// TwinCAT 3 PLC project PLC
// ProgramVersion: 3.1.4024.0
// libraries:
//   Tc2_Standard, * (Beckhoff Automation GmbH)
//   Tc2_System, * (Beckhoff Automation GmbH)
//   Tc3_Module, * (Beckhoff Automation GmbH)
// project tree:
//   DUTs/ FixtureInput.TcDUT, FixtureOutput.TcDUT, RollerDoor.TcDUT, Turn.TcDUT, TurnTableOutput.TcDUT
//   DUTs/Robot/ udt_HDL_CellToHandling.TcDUT, udt_HDL_HandlingToCell.TcDUT, udt_HDL_PartData.TcDUT
//   / GlobalTextList.TcGTLO, PlcTask.TcTTO, Visualization Manager.TcVMO (not stored)
//   GVLs/ IO.TcGVL, Memory.TcGVL, HMI.TcGVL, RobotInterface.TcGVL, WeldRobotInterface.TcGVL
//   POUs/ AutoSequence.TcPOU, Call_Fb.TcPOU, Feedback.TcPOU, Clamping.TcPOU, MAIN.TcPOU, RobotMH.TcPOU, RoolerDoor.TcPOU, Turn_Table.TcPOU, Turning_fb.TcPOU, vishalTest.TcPOU, WeldRobot.TcPOU
//   VISUs/ Clamp.TcVIS
// real-time tasks:
//   TASK PlcTask: cycle T#10ms, priority 20, ADS port 350

CONFIGURATION PLC
    RESOURCE PLC ON TwinCAT3
        TASK PlcTask(INTERVAL := T#10ms, PRIORITY := 20);
        PROGRAM MAIN WITH PlcTask : MAIN;
    END_RESOURCE
END_CONFIGURATION

// ---- DUTs/FixtureInput.TcDUT
TYPE FixtureInput :
STRUCT
i_Control_Pressure_Sw_In1_BPB1:BOOL;
i_Control_Pressure_Sw_In2_BPB1:BOOL;
i_Valve_Pos_BGB1:BOOL;
i_Reserve_BPB1_0_3:BOOL;
i_CC6_Clamp_1_Sensor_HP:BOOL;
i_CC6_Clamp_1_Sensor_WP:BOOL;
i_CC4_Clamp_3_Sensor_HP:BOOL;
i_CC4_Clamp_3_Sensor_WP:BOOL;
i_PART_CONTROL_B13:BOOL;
i_PART_CONTROL_B27:BOOL;
i_PART_CONTROL_B14:BOOL;
i_PART_CONTROL_B28:BOOL;
i_Reserve_BGB1_1_4:BOOL;
i_Reserve_BGB1_1_5:BOOL;

i_Reserve_2_0:BOOL;
i_Reserve_2_1:BOOL;
i_Reserve_2_2:BOOL;
i_Reserve_2_3:BOOL;
i_Reserve_2_4:BOOL;
i_Reserve_2_5:BOOL;
i_Reserve_2_6:BOOL;
i_Reserve_2_7:BOOL;
i_Reserve_3_0:BOOL;
i_Reserve_3_1:BOOL;
i_Reserve_3_2:BOOL;
i_Reserve_3_3:BOOL;
i_Reserve_3_4:BOOL;
i_Reserve_3_5:BOOL;
i_Reserve_3_6:BOOL;
i_Reserve_3_7:BOOL;
i_CC4_Clamp_2_Sensor_HP:BOOL;
i_CC4_Clamp_2_Sensor_WP:BOOL;
i_CC4_Clamp_1_Sensor_HP:BOOL;
i_CC4_Clamp_1_Sensor_WP:BOOL;
i_CC2_Clamp_3_Sensor_HP:BOOL;
i_CC2_Clamp_3_Sensor_WP:BOOL;
i_PART_CONTROL_B12:BOOL;
i_PART_CONTROL_B26:BOOL;
i_PART_CONTROL_B11:BOOL;
i_PART_CONTROL_B25:BOOL;
i_PART_CONTROL_B10:BOOL;
i_PART_CONTROL_B24:BOOL;
i_Reserve_5_4:BOOL;
i_Reserve_5_5:BOOL;
i_Reserve_5_6:BOOL;
i_Reserve_5_7:BOOL;
i_Reserve_6_0:BOOL;
i_Reserve_6_1:BOOL;
i_Reserve_6_2:BOOL;
i_Reserve_6_3:BOOL;
i_Reserve_6_4:BOOL;
i_Reserve_6_5:BOOL;
i_Reserve_6_6:BOOL;
i_Reserve_6_7:BOOL;
i_Reserve_7_1:BOOL;
i_Reserve_7_2:BOOL;
i_Reserve_7_3:BOOL;
i_Reserve_7_4:BOOL;
i_Reserve_7_5:BOOL;
i_Reserve_7_6:BOOL;
i_Reserve_7_7:BOOL;
i_CC3_Clamp_3_Sensor_HP:BOOL;
i_CC3_Clamp_3_Sensor_WP:BOOL;
i_CC3_Clamp_2_Sensor_HP:BOOL;
i_CC3_Clamp_2_Sensor_WP:BOOL;
i_CC3_Clamp_1_Sensor_HP:BOOL;
i_CC3_Clamp_1_Sensor_WP:BOOL;
i_PART_CONTROL_B7:BOOL;
i_PART_CONTROL_B21:BOOL;
i_PART_CONTROL_B6:BOOL;
i_PART_CONTROL_B20:BOOL;
i_PART_CONTROL_B5:BOOL;
i_PART_CONTROL_B19:BOOL;
i_Reserve_9_4:BOOL;
i_Reserve_9_5:BOOL;

i_CC1_Clamp_3_Sensor_HP:BOOL;
i_CC1_Clamp_3_Sensor_WP:BOOL;
i_CC1_Clamp_2_Sensor_HP:BOOL;
i_CC1_Clamp_2_Sensor_WP:BOOL;
i_CC1_Clamp_1_Sensor_HP:BOOL;
i_CC1_Clamp_1_Sensor_WP:BOOL;
i_PART_CONTROL_B4:BOOL;
i_PART_CONTROL_B18:BOOL;
i_PART_CONTROL_B3:BOOL;
i_PART_CONTROL_B17:BOOL;
i_PART_CONTROL_B2:BOOL;
i_PART_CONTROL_B16:BOOL;

i_CC2_Clamp_2_Sensor_HP:BOOL;
i_CC2_Clamp_2_Sensor_WP:BOOL;
i_CC2_Clamp_1_Sensor_HP:BOOL;
i_CC2_Clamp_1_Sensor_WP:BOOL;
i_PART_CONTROL_B9:BOOL;
i_PART_CONTROL_B23:BOOL;
i_PART_CONTROL_B8:BOOL;
i_PART_CONTROL_B22:BOOL;

i_CC5_Clamp_1_Sensor_HP:BOOL;
i_CC5_Clamp_1_Sensor_WP:BOOL;
i_PART_CONTROL_B1:BOOL;
i_PART_CONTROL_B15:BOOL;



END_STRUCT
END_TYPE

// ---- DUTs/FixtureOutput.TcDUT
TYPE FixtureOutput :
STRUCT
	o_CC1_CLAMPING_UNIT1_3_WP:BOOL;
o_CC1_CLAMPING_UNIT1_3_HP:BOOL;
o_CC2_CLAMPING_UNIT2_3_WP:BOOL;
o_CC2_CLAMPING_UNIT2_3_HP:BOOL;
o_CC3_CLAMPING_UNIT3_3_WP:BOOL;
o_CC3_CLAMPING_UNIT3_3_HP:BOOL;
o_CC4_CLAMPING_UNIT4_3_WP:BOOL;
o_CC4_CLAMPING_UNIT4_3_HP:BOOL;
o_CC5_CLAMPING_UNIT5_1_WP:BOOL;
o_CC5_CLAMPING_UNIT5_1_HP:BOOL;
o_CC6_CLAMPING_UNIT6_1_WP:BOOL;
o_CC6_CLAMPING_UNIT6_1_HP:BOOL;
o_RESERVE_1_4:BOOL;
o_RESERVE_1_5:BOOL;
o_RESERVE_1_6:BOOL;
o_RESERVE_1_7:BOOL;
o_RESERVE_2_0:BOOL;
o_RESERVE_2_1:BOOL;
o_RESERVE_2_2:BOOL;
o_RESERVE_2_3:BOOL;
o_RESERVE_2_4:BOOL;
o_RESERVE_2_5:BOOL;
o_RESERVE_2_6:BOOL;
o_RESERVE_2_7:BOOL;
o_RESERVE_3_0:BOOL;
o_RESERVE_3_1:BOOL;
o_RESERVE_3_2:BOOL;
o_RESERVE_3_3:BOOL;
o_RESERVE_3_4:BOOL;
o_RESERVE_3_5:BOOL;
o_RESERVE_3_6:BOOL;
o_RESERVE_3_7:BOOL;

END_STRUCT
END_TYPE

// ---- DUTs/Robot/udt_HDL_CellToHandling.TcDUT
TYPE udt_HDL_CellToHandling :
STRUCT
    (* Cell state *)
    Status      : WORD; // 0: Auto, 2: Manual, 3: Error
    Time_Stamp  : DATE_AND_TIME;
    part        : udt_HDL_PartData; // part
    
    (* Job Handshake *)
    Request             : USINT; // 20: Pick, 10: Drop
    RequestPartType     : BOOL;
    GateOpened          : BOOL;
    GateClosed          : BOOL;
    FixtureReady        : BOOL;
    (* Progress Feedback *)
	RaiseEnable1        : BOOL;
    RaiseEnable2        : BOOL;
    ReduceEnable1       : BOOL;
    ReduceEnable2       : BOOL;
     (* Status/Confirmation *)
	PickJobAck          : BOOL;
    DropJobAck          : BOOL;
    Hold                : BOOL;
    (* Gripper Acknowledge *)
	Gripper1ReadyToClose : BOOL;
    Gripper1ReadyToOpen  : BOOL;
    Gripper2ReadyToClose : BOOL;
    Gripper2ReadyToOpen  : BOOL;
    FeatureBit6         : BOOL;
    FeatureBit7         : BOOL;
END_STRUCT
END_TYPE

// ---- DUTs/Robot/udt_HDL_HandlingToCell.TcDUT
TYPE udt_HDL_HandlingToCell :
STRUCT
	
(* HDL Data *)
    Status      : WORD; // 0 Auto -- 1 Auto Startup -- 2 Manual -- 3 Error -- 4 LineMode -- 5 PowerOn -- 6 EnergySave -- 7 SafeOk
    part        : udt_HDL_PartData; // part
    
    (* Job Handshake Requests & Logic *)
    GateOpenRequest     : BOOL;
    GateCloseRequest    : BOOL;
    PickJobProceed      : BOOL;
    DropJobProceed      : BOOL;
    
    (* Progress Feedback *)
    RaiseFinished1      : BOOL;
    RaiseFinished2      : BOOL;
    ReduceFinished1     : BOOL;
    ReduceFinished2     : BOOL;
    
    (* Status/Confirmation *)
    PickJobOK           : BOOL;
    DropJobOK           : BOOL;
    InArea              : BOOL;
    PickDropProceed     : BOOL;
    
    (* Gripper Acknowledge *)
    Gripper1ClosedAck   : BOOL;
    Gripper1OpenedAck   : BOOL;
    Gripper2ClosedAck   : BOOL;
    Gripper2OpenedAck   : BOOL;
    
    (* Spare/Auxiliary *)
    FeatureBit6         : BOOL;
    FeatureBit7         : BOOL;
    PickEnable          : BOOL;
    DropEnable          : BOOL;
    
    (* Process Data *)
    Types               : USINT;
    ActiveCell          : USINT;
    Cooling_Time_Buffer : DINT;
    FB_Cooling_Time     : DINT;
END_STRUCT
END_TYPE

// ---- DUTs/Robot/udt_HDL_PartData.TcDUT
TYPE udt_HDL_PartData :
STRUCT
PartId	:DINT; //Unique Part Id (DMC Serial Number)
State	:BOOL; //Part state 0=OK, 1=NOK
Types :	BOOL;// Part type 1=Long, 0=Short
Exists	:BOOL; //Part exist


END_STRUCT
END_TYPE

// ---- DUTs/RollerDoor.TcDUT
TYPE RollerDoor :
STRUCT
	
i_RD_Sensor_Open:BOOL;
i_RD_Sensor_Close:BOOL;
o_RD_Open:BOOL;
o_RD_Close:BOOL;

END_STRUCT
END_TYPE

// ---- DUTs/Turn.TcDUT
TYPE Turn :
STRUCT
	o_Turn_REF_SENSOR:BOOL;
o_Turn_FWD_SENSOR:BOOL;
o_Turn_REV_SENSOR:BOOL;
END_STRUCT
END_TYPE

// ---- DUTs/TurnTableOutput.TcDUT
TYPE TurnTableOutput :
STRUCT
	
o_TurnTable_REF_SENSOR:BOOL;
o_TurnTable_FWD_SENSOR:BOOL;
o_TurnTable_REV_SENSOR:BOOL;
END_STRUCT

END_TYPE

// ---- GVLs/IO.TcGVL
{attribute 'qualified_only'}
VAR_GLOBAL
	FixtureInput:FixtureInput;
	FixtureOutput:FixtureOutput;
TurnTableOutput:TurnTableOutput;
Turn:Turn;
RD1:RollerDoor;
RD2:RollerDoor;
END_VAR

// ---- GVLs/Memory.TcGVL
{attribute 'qualified_only'}
VAR_GLOBAL

CC1_Clamp_FwdCmd:BOOL;
CC1_Clamp_RevCmd:BOOL;
CC2_Clamp_FwdCmd:BOOL;
CC2_Clamp_RevCmd:BOOL;
CC3_Clamp_FwdCmd:BOOL;
CC3_Clamp_RevCmd:BOOL;
CC4_Clamp_FwdCmd:BOOL;
CC4_Clamp_RevCmd:BOOL;
CC5_Clamp_FwdCmd:BOOL;
CC5_Clamp_RevCmd:BOOL;
CC6_Clamp_FwdCmd:BOOL;
CC6_Clamp_RevCmd:BOOL;
	
CC1_Clamp_Fwd:BOOL;
CC1_Clamp_Rev:BOOL;
CC2_Clamp_Fwd:BOOL;
CC2_Clamp_Rev:BOOL;
CC3_Clamp_Fwd:BOOL;
CC3_Clamp_Rev:BOOL;
CC4_Clamp_Fwd:BOOL;
CC4_Clamp_Rev:BOOL;
CC5_Clamp_Fwd:BOOL;
CC5_Clamp_Rev:BOOL;
CC6_Clamp_Fwd:BOOL;
CC6_Clamp_Rev:BOOL;
AllClampWP:BOOL;
AllClampHP:BOOL;


TurnTableRef:BOOL;
TurnTableRefDone:BOOL;
TurnTableFwdCmd:BOOL;
TurnTableFwd:BOOL;
TurnTableRevCmd:BOOL;
TurnTableRev:BOOL;


TurnRef:BOOL;
TurnRefDone:BOOL;
TurnFwdCmd:BOOL;
TurnFwd:BOOL;
TurnRevCmd:BOOL;
TurnRev:BOOL;

RD1_OpenCmd:BOOL;
RD1_CloseCmd:BOOL;
RD1_Open:BOOL;
RD1_Close:BOOL;
RD2_OpenCmd:BOOL;
RD2_CloseCmd:BOOL;
RD2_Open:BOOL;
RD2_Close:BOOL;

Stat_Parts_Lvl1_Present:BOOL;
Stat_Parts_Lvl2_Present:BOOL;
In_PalmButton_Pushed:BOOL;
In_Welding_Cycle_Complete:BOOL;
In_Operator_Outside_Cell:BOOL;
In_Operator_Inside_Cell:BOOL;
Out_Robot_Start_Unload_1:BOOL;
Out_Robot_Start_Unload_2:BOOL;

AutoMode:BOOL;
ManualMode:BOOL;
END_VAR

// ---- GVLs/HMI.TcGVL
{attribute 'qualified_only'}
VAR_GLOBAL

CC1_Clamp_FwdCmd:BOOL;
CC1_Clamp_RevCmd:BOOL;
CC2_Clamp_FwdCmd:BOOL;
CC2_Clamp_RevCmd:BOOL;
CC3_Clamp_FwdCmd:BOOL;
CC3_Clamp_RevCmd:BOOL;
CC4_Clamp_FwdCmd:BOOL;
CC4_Clamp_RevCmd:BOOL;
CC5_Clamp_FwdCmd:BOOL;
CC5_Clamp_RevCmd:BOOL;
CC6_Clamp_FwdCmd:BOOL;
CC6_Clamp_RevCmd:BOOL;
	
CC1_Clamp_Fwd:BOOL;
CC1_Clamp_Rev:BOOL;
CC2_Clamp_Fwd:BOOL;
CC2_Clamp_Rev:BOOL;
CC3_Clamp_Fwd:BOOL;
CC3_Clamp_Rev:BOOL;
CC4_Clamp_Fwd:BOOL;
CC4_Clamp_Rev:BOOL;
CC5_Clamp_Fwd:BOOL;
CC5_Clamp_Rev:BOOL;
CC6_Clamp_Fwd:BOOL;
CC6_Clamp_Rev:BOOL;

TurnTableRef:BOOL;
TurnTableRefDone:BOOL;
TurnTableFwdCmd:BOOL;
TurnTableFwd:BOOL;
TurnTableRevCmd:BOOL;
TurnTableRev:BOOL;


TurnRef:BOOL;
TurnRefDone:BOOL;
TurnFwdCmd:BOOL;
TurnFwd:BOOL;
TurnRevCmd:BOOL;
TurnRev:BOOL;

RD1_OpenCmd:BOOL;
RD1_CloseCmd:BOOL;
RD1_Open:BOOL;
RD1_Close:BOOL;
RD2_OpenCmd:BOOL;
RD2_CloseCmd:BOOL;
RD2_Open:BOOL;
RD2_Close:BOOL;

Stat_Parts_Lvl1_Present:BOOL;
Stat_Parts_Lvl2_Present:BOOL;
In_PalmButton_Pushed:BOOL;
In_Welding_Cycle_Complete:BOOL;
In_Operator_Outside_Cell:BOOL;
In_Operator_Inside_Cell:BOOL;
Out_Robot_Start_Unload_1:BOOL;
Out_Robot_Start_Unload_2:BOOL;

AutoMode:BOOL;
ManualMode:BOOL;
Home:BOOL;
ReadyForLoad:BOOL;
END_VAR

// ---- GVLs/RobotInterface.TcGVL
{attribute 'qualified_only'}
VAR_GLOBAL
	HDL_CellToHandling:udt_HDL_CellToHandling;
	HDL_HandlingToCell:udt_HDL_HandlingToCell;
RobotAtPickPosition:BOOL;
RobotAtDropPosition:BOOL;
RobotAtHome:BOOL;



END_VAR

// ---- GVLs/WeldRobotInterface.TcGVL
{attribute 'qualified_only'}
VAR_GLOBAL
	CellToWeld:udt_HDL_CellToHandling;
	WeldToCell:udt_HDL_HandlingToCell;
RobotAtWeldPosition:BOOL;
RobotAtDropPosition:BOOL;
RobotAtHome:BOOL;
TorchOn:bool;


END_VAR

// ---- POUs/MAIN.TcPOU
PROGRAM MAIN
VAR
	
	Call_Fb_Idb: Call_Fb;
	Fixture_Idb: Clamping;
END_VAR

Call_Fb_Idb();

Fixture_Idb();

END_PROGRAM

// ---- POUs/Call_Fb.TcPOU
FUNCTION_BLOCK Call_Fb
VAR_INPUT
END_VAR
VAR_OUTPUT
END_VAR
VAR
	Feedback_CC1_Clamp1: Feedback;
	Feedback_CC1_Clamp2: Feedback;
	Feedback_CC1_Clamp3: Feedback;
	Feedback_CC2_Clamp1: Feedback;
	Feedback_CC2_Clamp2: Feedback;
	Feedback_CC2_Clamp3: Feedback;
	Feedback_CC3_Clamp1: Feedback;
	Feedback_CC3_Clamp2: Feedback;
	Feedback_CC3_Clamp3: Feedback;
	Feedback_CC4_Clamp1: Feedback;
	Feedback_CC4_Clamp2: Feedback;
	Feedback_CC4_Clamp3: Feedback;
	Feedback_CC5_Clamp1: Feedback;
	Feedback_CC6_Clamp1: Feedback;

	Feedback_TT: Feedback;
	Feedback_TT1: Feedback;
	Turn_Table_0: Turn_Table;

		Turning_fb_0: Turning_fb;
	Feedback_Turn: Feedback;
	Feedback_Turn1: Feedback;
	RoolerDoor_1: RoolerDoor;
	Feedback_RD1: Feedback;
	RoolerDoor_2: RoolerDoor;
	Feedback_RD2: Feedback;
	Robot_MH: RobotMH;
	AutoSequence_0: AutoSequence;
	WeldRobot_0: WeldRobot;
	
END_VAR

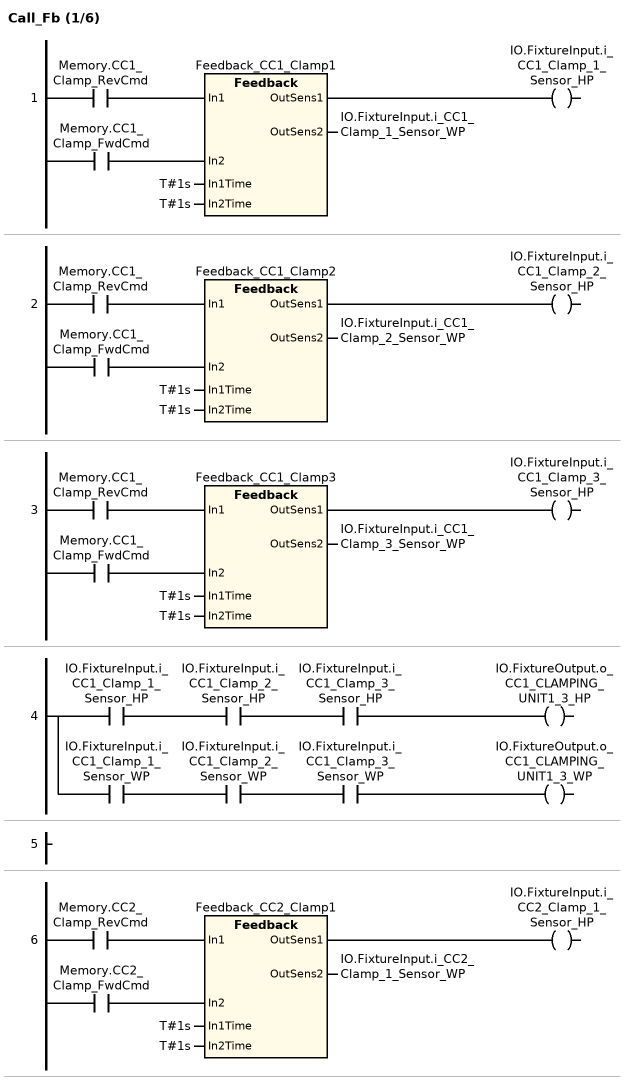
// NETWORK 1
Feedback_CC1_Clamp1(
    In1 := Memory.CC1_Clamp_RevCmd,
    In2 := Memory.CC1_Clamp_FwdCmd,
    In1Time := T#1s,
    In2Time := T#1s,
    OutSens2 => IO.FixtureInput.i_CC1_Clamp_1_Sensor_WP); // Feedback
IO.FixtureInput.i_CC1_Clamp_1_Sensor_HP := Feedback_CC1_Clamp1.OutSens1;

// NETWORK 2
Feedback_CC1_Clamp2(
    In1 := Memory.CC1_Clamp_RevCmd,
    In2 := Memory.CC1_Clamp_FwdCmd,
    In1Time := T#1s,
    In2Time := T#1s,
    OutSens2 => IO.FixtureInput.i_CC1_Clamp_2_Sensor_WP); // Feedback
IO.FixtureInput.i_CC1_Clamp_2_Sensor_HP := Feedback_CC1_Clamp2.OutSens1;

// NETWORK 3
Feedback_CC1_Clamp3(
    In1 := Memory.CC1_Clamp_RevCmd,
    In2 := Memory.CC1_Clamp_FwdCmd,
    In1Time := T#1s,
    In2Time := T#1s,
    OutSens2 => IO.FixtureInput.i_CC1_Clamp_3_Sensor_WP); // Feedback
IO.FixtureInput.i_CC1_Clamp_3_Sensor_HP := Feedback_CC1_Clamp3.OutSens1;

// NETWORK 4
IO.FixtureOutput.o_CC1_CLAMPING_UNIT1_3_HP := IO.FixtureInput.i_CC1_Clamp_1_Sensor_HP AND IO.FixtureInput.i_CC1_Clamp_2_Sensor_HP AND IO.FixtureInput.i_CC1_Clamp_3_Sensor_HP;
IO.FixtureOutput.o_CC1_CLAMPING_UNIT1_3_WP := IO.FixtureInput.i_CC1_Clamp_1_Sensor_WP AND IO.FixtureInput.i_CC1_Clamp_2_Sensor_WP AND IO.FixtureInput.i_CC1_Clamp_3_Sensor_WP;

// NETWORK 5

// NETWORK 6
Feedback_CC2_Clamp1(
    In1 := Memory.CC2_Clamp_RevCmd,
    In2 := Memory.CC2_Clamp_FwdCmd,
    In1Time := T#1s,
    In2Time := T#1s,
    OutSens2 => IO.FixtureInput.i_CC2_Clamp_1_Sensor_WP); // Feedback
IO.FixtureInput.i_CC2_Clamp_1_Sensor_HP := Feedback_CC2_Clamp1.OutSens1;

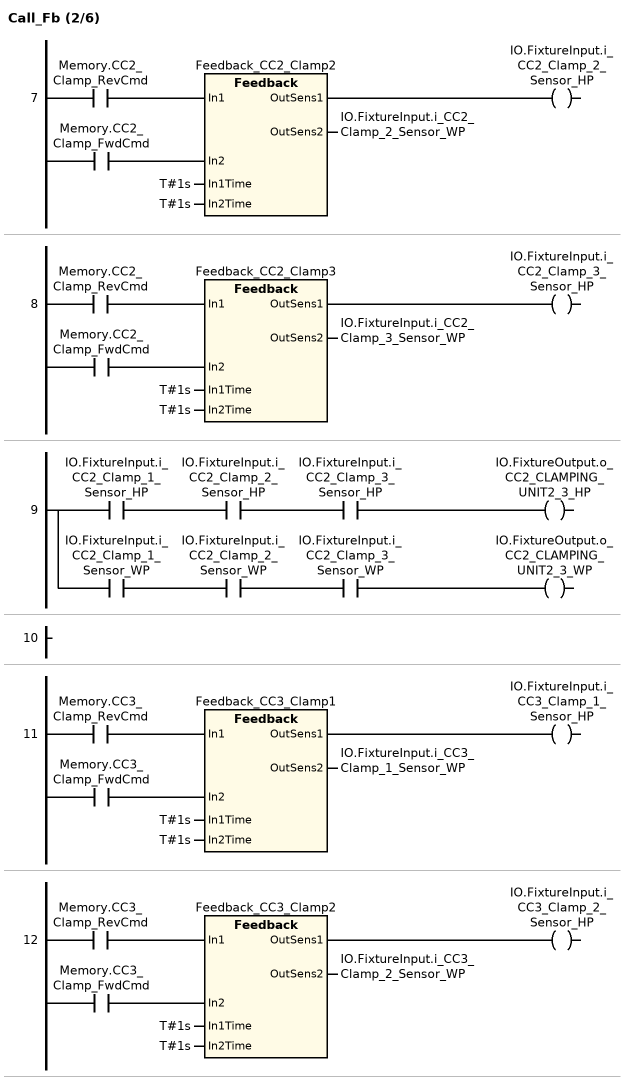
// NETWORK 7
Feedback_CC2_Clamp2(
    In1 := Memory.CC2_Clamp_RevCmd,
    In2 := Memory.CC2_Clamp_FwdCmd,
    In1Time := T#1s,
    In2Time := T#1s,
    OutSens2 => IO.FixtureInput.i_CC2_Clamp_2_Sensor_WP); // Feedback
IO.FixtureInput.i_CC2_Clamp_2_Sensor_HP := Feedback_CC2_Clamp2.OutSens1;

// NETWORK 8
Feedback_CC2_Clamp3(
    In1 := Memory.CC2_Clamp_RevCmd,
    In2 := Memory.CC2_Clamp_FwdCmd,
    In1Time := T#1s,
    In2Time := T#1s,
    OutSens2 => IO.FixtureInput.i_CC2_Clamp_3_Sensor_WP); // Feedback
IO.FixtureInput.i_CC2_Clamp_3_Sensor_HP := Feedback_CC2_Clamp3.OutSens1;

// NETWORK 9
IO.FixtureOutput.o_CC2_CLAMPING_UNIT2_3_HP := IO.FixtureInput.i_CC2_Clamp_1_Sensor_HP AND IO.FixtureInput.i_CC2_Clamp_2_Sensor_HP AND IO.FixtureInput.i_CC2_Clamp_3_Sensor_HP;
IO.FixtureOutput.o_CC2_CLAMPING_UNIT2_3_WP := IO.FixtureInput.i_CC2_Clamp_1_Sensor_WP AND IO.FixtureInput.i_CC2_Clamp_2_Sensor_WP AND IO.FixtureInput.i_CC2_Clamp_3_Sensor_WP;

// NETWORK 10

// NETWORK 11
Feedback_CC3_Clamp1(
    In1 := Memory.CC3_Clamp_RevCmd,
    In2 := Memory.CC3_Clamp_FwdCmd,
    In1Time := T#1s,
    In2Time := T#1s,
    OutSens2 => IO.FixtureInput.i_CC3_Clamp_1_Sensor_WP); // Feedback
IO.FixtureInput.i_CC3_Clamp_1_Sensor_HP := Feedback_CC3_Clamp1.OutSens1;

// NETWORK 12
Feedback_CC3_Clamp2(
    In1 := Memory.CC3_Clamp_RevCmd,
    In2 := Memory.CC3_Clamp_FwdCmd,
    In1Time := T#1s,
    In2Time := T#1s,
    OutSens2 => IO.FixtureInput.i_CC3_Clamp_2_Sensor_WP); // Feedback
IO.FixtureInput.i_CC3_Clamp_2_Sensor_HP := Feedback_CC3_Clamp2.OutSens1;

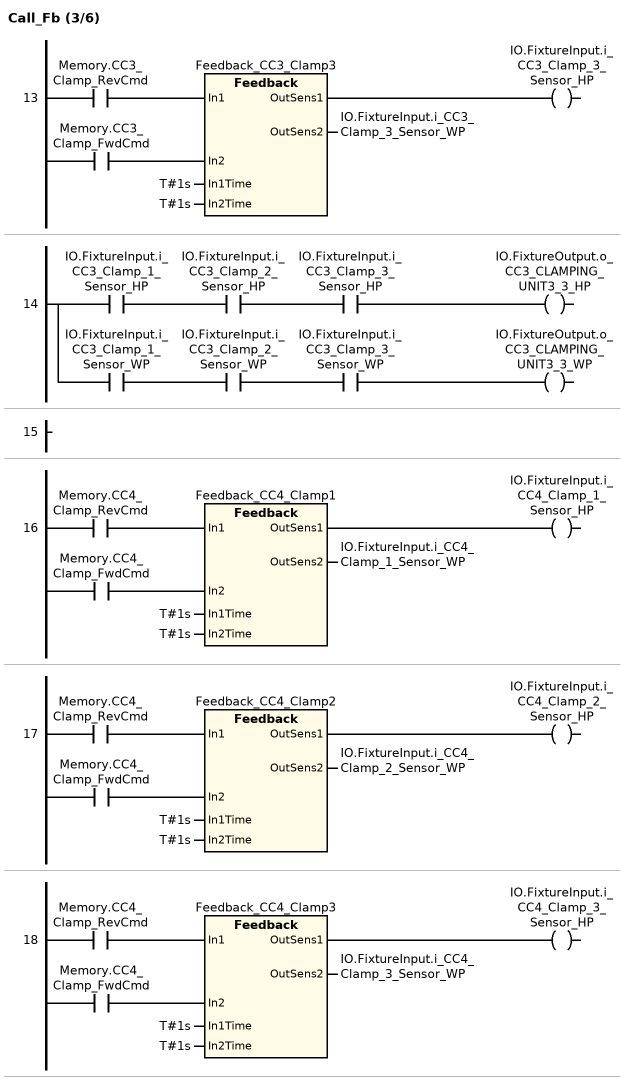
// NETWORK 13
Feedback_CC3_Clamp3(
    In1 := Memory.CC3_Clamp_RevCmd,
    In2 := Memory.CC3_Clamp_FwdCmd,
    In1Time := T#1s,
    In2Time := T#1s,
    OutSens2 => IO.FixtureInput.i_CC3_Clamp_3_Sensor_WP); // Feedback
IO.FixtureInput.i_CC3_Clamp_3_Sensor_HP := Feedback_CC3_Clamp3.OutSens1;

// NETWORK 14
IO.FixtureOutput.o_CC3_CLAMPING_UNIT3_3_HP := IO.FixtureInput.i_CC3_Clamp_1_Sensor_HP AND IO.FixtureInput.i_CC3_Clamp_2_Sensor_HP AND IO.FixtureInput.i_CC3_Clamp_3_Sensor_HP;
IO.FixtureOutput.o_CC3_CLAMPING_UNIT3_3_WP := IO.FixtureInput.i_CC3_Clamp_1_Sensor_WP AND IO.FixtureInput.i_CC3_Clamp_2_Sensor_WP AND IO.FixtureInput.i_CC3_Clamp_3_Sensor_WP;

// NETWORK 15

// NETWORK 16
Feedback_CC4_Clamp1(
    In1 := Memory.CC4_Clamp_RevCmd,
    In2 := Memory.CC4_Clamp_FwdCmd,
    In1Time := T#1s,
    In2Time := T#1s,
    OutSens2 => IO.FixtureInput.i_CC4_Clamp_1_Sensor_WP); // Feedback
IO.FixtureInput.i_CC4_Clamp_1_Sensor_HP := Feedback_CC4_Clamp1.OutSens1;

// NETWORK 17
Feedback_CC4_Clamp2(
    In1 := Memory.CC4_Clamp_RevCmd,
    In2 := Memory.CC4_Clamp_FwdCmd,
    In1Time := T#1s,
    In2Time := T#1s,
    OutSens2 => IO.FixtureInput.i_CC4_Clamp_2_Sensor_WP); // Feedback
IO.FixtureInput.i_CC4_Clamp_2_Sensor_HP := Feedback_CC4_Clamp2.OutSens1;

// NETWORK 18
Feedback_CC4_Clamp3(
    In1 := Memory.CC4_Clamp_RevCmd,
    In2 := Memory.CC4_Clamp_FwdCmd,
    In1Time := T#1s,
    In2Time := T#1s,
    OutSens2 => IO.FixtureInput.i_CC4_Clamp_3_Sensor_WP); // Feedback
IO.FixtureInput.i_CC4_Clamp_3_Sensor_HP := Feedback_CC4_Clamp3.OutSens1;

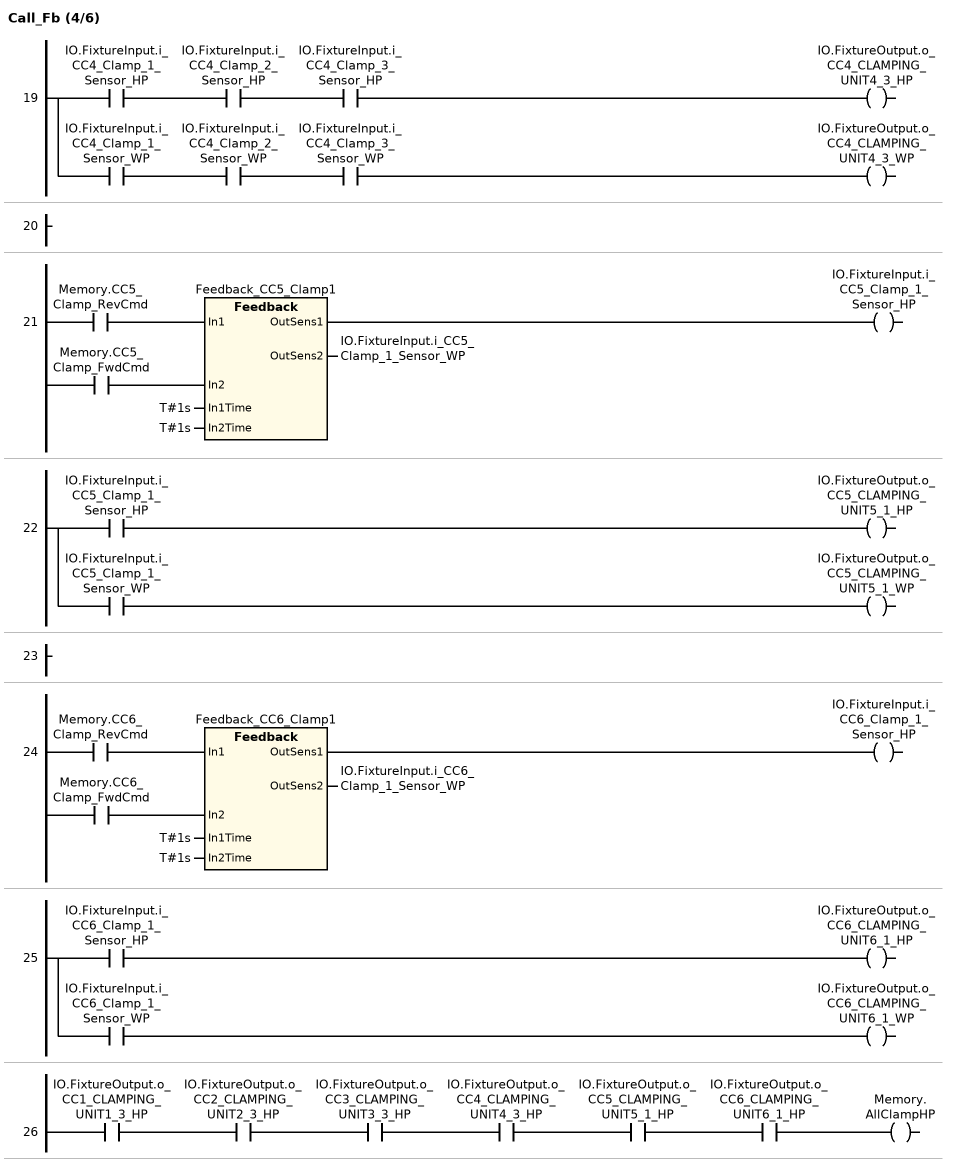
// NETWORK 19
IO.FixtureOutput.o_CC4_CLAMPING_UNIT4_3_HP := IO.FixtureInput.i_CC4_Clamp_1_Sensor_HP AND IO.FixtureInput.i_CC4_Clamp_2_Sensor_HP AND IO.FixtureInput.i_CC4_Clamp_3_Sensor_HP;
IO.FixtureOutput.o_CC4_CLAMPING_UNIT4_3_WP := IO.FixtureInput.i_CC4_Clamp_1_Sensor_WP AND IO.FixtureInput.i_CC4_Clamp_2_Sensor_WP AND IO.FixtureInput.i_CC4_Clamp_3_Sensor_WP;

// NETWORK 20

// NETWORK 21
Feedback_CC5_Clamp1(
    In1 := Memory.CC5_Clamp_RevCmd,
    In2 := Memory.CC5_Clamp_FwdCmd,
    In1Time := T#1s,
    In2Time := T#1s,
    OutSens2 => IO.FixtureInput.i_CC5_Clamp_1_Sensor_WP); // Feedback
IO.FixtureInput.i_CC5_Clamp_1_Sensor_HP := Feedback_CC5_Clamp1.OutSens1;

// NETWORK 22
IO.FixtureOutput.o_CC5_CLAMPING_UNIT5_1_HP := IO.FixtureInput.i_CC5_Clamp_1_Sensor_HP;
IO.FixtureOutput.o_CC5_CLAMPING_UNIT5_1_WP := IO.FixtureInput.i_CC5_Clamp_1_Sensor_WP;

// NETWORK 23

// NETWORK 24
Feedback_CC6_Clamp1(
    In1 := Memory.CC6_Clamp_RevCmd,
    In2 := Memory.CC6_Clamp_FwdCmd,
    In1Time := T#1s,
    In2Time := T#1s,
    OutSens2 => IO.FixtureInput.i_CC6_Clamp_1_Sensor_WP); // Feedback
IO.FixtureInput.i_CC6_Clamp_1_Sensor_HP := Feedback_CC6_Clamp1.OutSens1;

// NETWORK 25
IO.FixtureOutput.o_CC6_CLAMPING_UNIT6_1_HP := IO.FixtureInput.i_CC6_Clamp_1_Sensor_HP;
IO.FixtureOutput.o_CC6_CLAMPING_UNIT6_1_WP := IO.FixtureInput.i_CC6_Clamp_1_Sensor_WP;

// NETWORK 26
Memory.AllClampHP := IO.FixtureOutput.o_CC1_CLAMPING_UNIT1_3_HP AND IO.FixtureOutput.o_CC2_CLAMPING_UNIT2_3_HP AND IO.FixtureOutput.o_CC3_CLAMPING_UNIT3_3_HP AND IO.FixtureOutput.o_CC4_CLAMPING_UNIT4_3_HP AND IO.FixtureOutput.o_CC5_CLAMPING_UNIT5_1_HP AND IO.FixtureOutput.o_CC6_CLAMPING_UNIT6_1_HP;

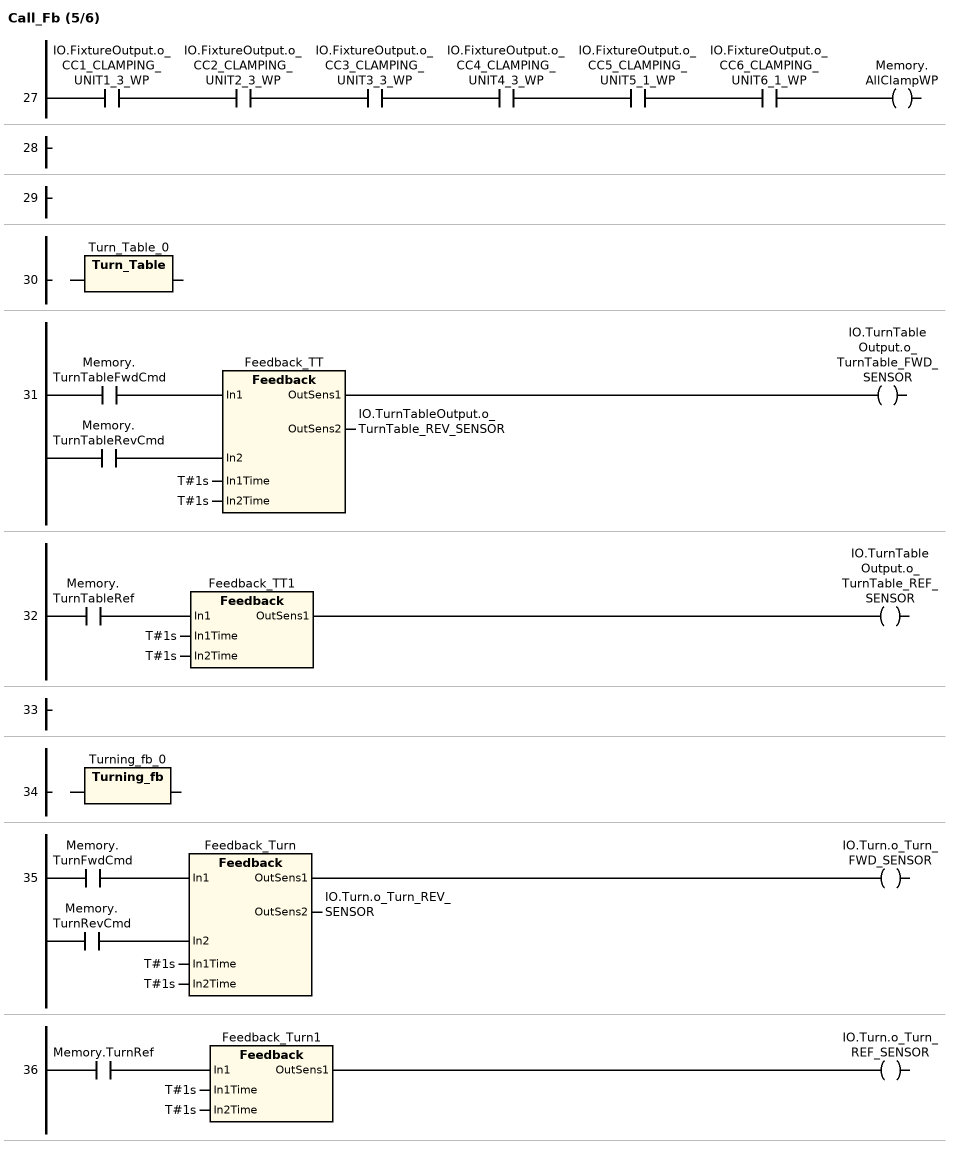
// NETWORK 27
Memory.AllClampWP := IO.FixtureOutput.o_CC1_CLAMPING_UNIT1_3_WP AND IO.FixtureOutput.o_CC2_CLAMPING_UNIT2_3_WP AND IO.FixtureOutput.o_CC3_CLAMPING_UNIT3_3_WP AND IO.FixtureOutput.o_CC4_CLAMPING_UNIT4_3_WP AND IO.FixtureOutput.o_CC5_CLAMPING_UNIT5_1_WP AND IO.FixtureOutput.o_CC6_CLAMPING_UNIT6_1_WP;

// NETWORK 28

// NETWORK 29

// NETWORK 30
Turn_Table_0(); // Turn_Table

// NETWORK 31
Feedback_TT(
    In1 := Memory.TurnTableFwdCmd,
    In2 := Memory.TurnTableRevCmd,
    In1Time := T#1s,
    In2Time := T#1s,
    OutSens2 => IO.TurnTableOutput.o_TurnTable_REV_SENSOR); // Feedback
IO.TurnTableOutput.o_TurnTable_FWD_SENSOR := Feedback_TT.OutSens1;

// NETWORK 32
Feedback_TT1(In1 := Memory.TurnTableRef, In1Time := T#1s, In2Time := T#1s); // Feedback
IO.TurnTableOutput.o_TurnTable_REF_SENSOR := Feedback_TT1.OutSens1;

// NETWORK 33

// NETWORK 34
Turning_fb_0(); // Turning_fb

// NETWORK 35
Feedback_Turn(
    In1 := Memory.TurnFwdCmd,
    In2 := Memory.TurnRevCmd,
    In1Time := T#1s,
    In2Time := T#1s,
    OutSens2 => IO.Turn.o_Turn_REV_SENSOR); // Feedback
IO.Turn.o_Turn_FWD_SENSOR := Feedback_Turn.OutSens1;

// NETWORK 36
Feedback_Turn1(In1 := Memory.TurnRef, In1Time := T#1s, In2Time := T#1s); // Feedback
IO.Turn.o_Turn_REF_SENSOR := Feedback_Turn1.OutSens1;

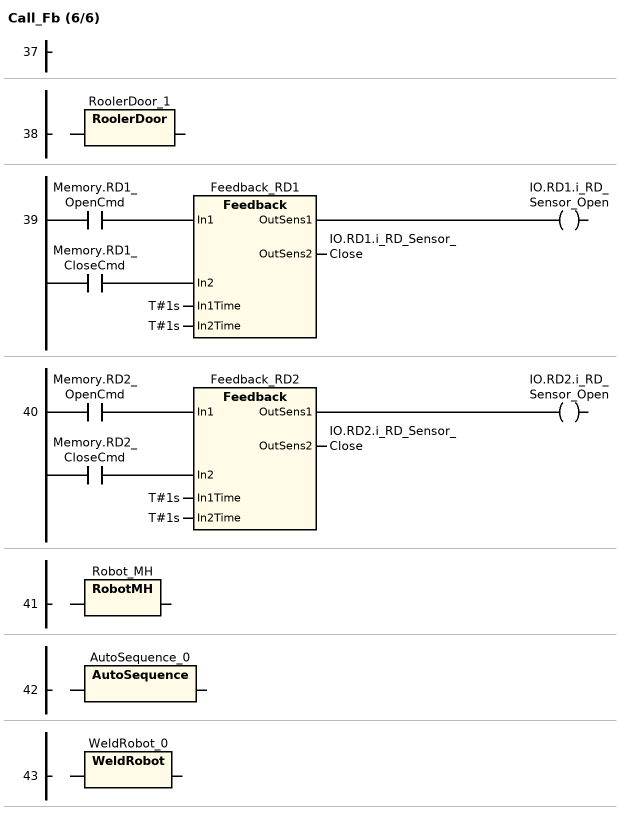
// NETWORK 37

// NETWORK 38
RoolerDoor_1(); // RoolerDoor

// NETWORK 39
Feedback_RD1(
    In1 := Memory.RD1_OpenCmd,
    In2 := Memory.RD1_CloseCmd,
    In1Time := T#1s,
    In2Time := T#1s,
    OutSens2 => IO.RD1.i_RD_Sensor_Close); // Feedback
IO.RD1.i_RD_Sensor_Open := Feedback_RD1.OutSens1;

// NETWORK 40
Feedback_RD2(
    In1 := Memory.RD2_OpenCmd,
    In2 := Memory.RD2_CloseCmd,
    In1Time := T#1s,
    In2Time := T#1s,
    OutSens2 => IO.RD2.i_RD_Sensor_Close); // Feedback
IO.RD2.i_RD_Sensor_Open := Feedback_RD2.OutSens1;

// NETWORK 41
Robot_MH(); // RobotMH

// NETWORK 42
AutoSequence_0(); // AutoSequence

// NETWORK 43
WeldRobot_0(); // WeldRobot

END_FUNCTION_BLOCK

// ---- POUs/Feedback.TcPOU
FUNCTION_BLOCK Feedback
VAR_INPUT
	In1:BOOL;
	In2:BOOL;
	In1Time:TIME;
	In2Time:TIME;
END_VAR
VAR_OUTPUT
	OutSens1:BOOL;
	OutSens2: BOOL;
END_VAR
VAR
	
	SenserDelay1: TON;
	SenserDelay2: TON;
END_VAR

// Sensor 1 logic
SenserDelay1(IN := In1, PT := In1Time);
IF SenserDelay1.Q THEN
    OutSens1 := TRUE;   // Output TurnTables ON after set seconds
	 OutSens2 := FALSE;
END_IF;

// Sensor 2 logic
SenserDelay2(IN := In2, PT := In2Time);
IF SenserDelay2.Q THEN
    OutSens2 := TRUE;   // Output TurnTables ON after set seconds
	OutSens1 := FALSE;
END_IF;

END_FUNCTION_BLOCK

// ---- POUs/Turn_Table.TcPOU
FUNCTION_BLOCK Turn_Table
VAR_INPUT
END_VAR
VAR_OUTPUT
END_VAR
VAR
END_VAR

// Homing sequence
IF NOT Memory.TurnTableRefDone OR Memory.TurnTableRef THEN
    Memory.TurnTableFwdCmd := TRUE;   // drive forward until reference
    IF IO.TurnTableOutput.o_TurnTable_REF_SENSOR THEN
        Memory.TurnTableFwdCmd := FALSE;
        Memory.TurnTableRefDone := TRUE;   // reference complete
    END_IF;
END_IF;

// Forward rotation
IF Memory.TurnTableFwdCmd AND Memory.TurnTableRefDone THEN
    Memory.TurnTableRev := FALSE;   // interlock
END_IF;

IF IO.TurnTableOutput.o_TurnTable_FWD_SENSOR THEN
    Memory.TurnTableFwd := TRUE;
END_IF;

// Reverse rotation
IF Memory.TurnTableRevCmd AND Memory.TurnTableRefDone THEN
    Memory.TurnTableFwd := FALSE;   // interlock
END_IF;

IF IO.TurnTableOutput.o_TurnTable_REV_SENSOR THEN
    Memory.TurnTableRev := TRUE;
END_IF;

END_FUNCTION_BLOCK

// ---- POUs/Turning_fb.TcPOU
FUNCTION_BLOCK Turning_fb
VAR_INPUT
END_VAR
VAR_OUTPUT
END_VAR
VAR
END_VAR

// Homing sequence
IF NOT Memory.TurnRefDone OR Memory.TurnTableRef THEN
    Memory.TurnFwdCmd := TRUE;   // drive forward until reference
    IF IO.Turn.o_Turn_REF_SENSOR THEN
        Memory.TurnFwdCmd := FALSE;
        Memory.TurnRefDone := TRUE;   // reference complete
    END_IF;
END_IF;

// Forward rotation work 50 deg
IF Memory.TurnFwdCmd AND Memory.TurnRefDone THEN
    Memory.TurnRev := FALSE;   // interlock
END_IF;

IF IO.Turn.o_Turn_FWD_SENSOR THEN
    Memory.TurnFwd := TRUE;
END_IF;

// Reverse rotation home 0 deg
IF Memory.TurnRevCmd AND Memory.TurnRefDone THEN
    Memory.TurnFwd := FALSE;   // interlock
END_IF;

IF IO.Turn.o_Turn_REV_SENSOR THEN
    Memory.TurnRev := TRUE;
END_IF;

END_FUNCTION_BLOCK

// ---- POUs/RoolerDoor.TcPOU
FUNCTION_BLOCK RoolerDoor
VAR_INPUT
END_VAR
VAR_OUTPUT
END_VAR
VAR
END_VAR

// Roller Door
IF Memory.RD1_OpenCmd OR RobotInterface.HDL_HandlingToCell.GateOpenRequest THEN
    Memory.RD1_Close := FALSE;
ELSIF Memory.RD1_CloseCmd OR RobotInterface.HDL_HandlingToCell.GateCloseRequest THEN
    Memory.RD1_Open := FALSE;
END_IF;

IF IO.RD1.i_RD_Sensor_Open THEN
    Memory.RD1_Open := TRUE;
END_IF;

IF IO.RD1.i_RD_Sensor_Close  THEN
    Memory.RD1_Close := TRUE;
END_IF;

// Roller Door 2
IF Memory.RD2_OpenCmd THEN
    Memory.RD2_Close := FALSE;
ELSIF Memory.RD2_CloseCmd THEN
    Memory.RD2_Open := FALSE;
END_IF;

IF IO.RD2.i_RD_Sensor_Open THEN//opened
    Memory.RD2_Open := TRUE;
END_IF;

IF IO.RD2.i_RD_Sensor_Close  THEN//closed
    Memory.RD2_Close := TRUE;
END_IF;

END_FUNCTION_BLOCK

// ---- POUs/RobotMH.TcPOU
FUNCTION_BLOCK RobotMH
VAR_INPUT
END_VAR
VAR_OUTPUT
END_VAR
VAR
    tGateOpen : TON;
    tDoorWait : TON;
    tGripClose : TON;
    tGripOpen : TON;
    tDropWait : TON;
    tReturnHome : TON;
	nState: INT;
	CycleCount : INT := 0;
END_VAR


IF Memory.AutoMode THEN
CASE nState OF

    0: (* WAIT FOR PART & PERMISSION *)
        RobotInterface.RobotAtHome := TRUE;
        RobotInterface.HDL_HandlingToCell.PickJobOK := FALSE;
        RobotInterface.HDL_HandlingToCell.Gripper1ClosedAck := FALSE;
        RobotInterface.HDL_HandlingToCell.Gripper1OpenedAck := TRUE;

        IF Memory.In_Welding_Cycle_Complete 
           AND WeldRobotInterface.RobotAtHome 
           AND IO.RD1.i_RD_Sensor_Open 
           AND (Memory.Stat_Parts_Lvl1_Present OR Memory.Stat_Parts_Lvl2_Present) THEN
            RobotInterface.HDL_HandlingToCell.PickEnable := TRUE;
            RobotInterface.HDL_HandlingToCell.InArea := TRUE;
            RobotInterface.HDL_HandlingToCell.PickDropProceed := TRUE;
            nState := 10;
        END_IF;

    10: (* GRIPPER ACTION *)
        RobotInterface.HDL_HandlingToCell.PickJobProceed := TRUE;
        tGripClose(IN := NOT tGripClose.q, PT := T#2S);
        RobotInterface.HDL_HandlingToCell.Gripper1ClosedAck := TRUE;
        RobotInterface.HDL_HandlingToCell.Gripper1OpenedAck := FALSE;
        RobotInterface.RobotAtHome := FALSE;

        IF tGripClose.Q THEN
            nState := 20;
        END_IF;

    20: (* VERIFY GRIPPER & CLEARANCE *)
        IF RobotInterface.HDL_HandlingToCell.Gripper1ClosedAck THEN
            RobotInterface.HDL_HandlingToCell.PickJobProceed := FALSE;
            RobotInterface.HDL_HandlingToCell.PickEnable := FALSE;
            RobotInterface.HDL_HandlingToCell.PickJobOK := TRUE;
            RobotInterface.HDL_HandlingToCell.InArea := FALSE;
            RobotInterface.HDL_HandlingToCell.DropEnable := TRUE;

            IF Memory.Out_Robot_Start_Unload_1 AND IO.Turn.o_Turn_REV_SENSOR THEN
                Memory.Stat_Parts_Lvl1_Present := FALSE;
            END_IF;
            IF Memory.Out_Robot_Start_Unload_2 AND IO.Turn.o_Turn_FWD_SENSOR THEN
                Memory.Stat_Parts_Lvl2_Present := FALSE;
            END_IF;

            IF NOT Memory.Stat_Parts_Lvl1_Present OR NOT Memory.Stat_Parts_Lvl2_Present THEN
                nState := 30;
            END_IF;
        END_IF;

    30: (* WAIT FOR PART & PERMISSION OF DROP *)
        IF RobotInterface.HDL_HandlingToCell.DropEnable AND NOT RobotInterface.HDL_HandlingToCell.DropJobOK THEN
            RobotInterface.HDL_HandlingToCell.InArea := TRUE;
            tDropWait(IN := NOT tDropWait.q, PT := T#2S);
            IF tDropWait.Q THEN
                nState := 40;
           END_IF;
        END_IF;

    40: (* WAIT FOR DROP *)
        IF RobotInterface.HDL_HandlingToCell.InArea AND RobotInterface.HDL_HandlingToCell.PickDropProceed THEN
            tDropWait(IN := FALSE);
            nState := 50;
        END_IF;

    50: (* GRIPPER ACTION *)
        RobotInterface.HDL_HandlingToCell.DropJobProceed := TRUE;
        tGripOpen(IN := TRUE, PT := T#2S);
        RobotInterface.HDL_HandlingToCell.Gripper1OpenedAck := TRUE;
        RobotInterface.HDL_HandlingToCell.Gripper1ClosedAck := FALSE;
        nState := 60;

    60: (* VERIFY GRIPPER & CLEARANCE *)
        IF RobotInterface.HDL_HandlingToCell.Gripper1OpenedAck THEN
            RobotInterface.HDL_HandlingToCell.DropJobProceed := FALSE;
            tReturnHome(IN := NOT tReturnHome.Q, PT := T#1S);
       IF tReturnHome.Q THEN
		  nState := 70;
	END_IF;
            RobotInterface.RobotAtHome := TRUE;
            RobotInterface.HDL_HandlingToCell.InArea := FALSE;
        END_IF;

    70: (* JOB COMPLETE *)
        RobotInterface.HDL_HandlingToCell.PickJobOK := TRUE;

        CycleCount := CycleCount + 1; // increment cycle count

        IF CycleCount < 2 THEN
            nState := 0; // repeat pick-drop
        ELSE
            CycleCount := 0; // reset after 2 cycles
            nState := 0;     // or go to idle state
        END_IF;

END_CASE;

ELSE

// Manual homing logic
IF HMI.Home THEN
    RobotInterface.RobotAtHome := TRUE;
    RobotInterface.HDL_HandlingToCell.Gripper1OpenedAck := TRUE;
    RobotInterface.HDL_HandlingToCell.Gripper1ClosedAck := FALSE;
    RobotInterface.HDL_HandlingToCell.InArea := FALSE;
    nState := 0; // reset state machine to idle
END_IF;
END_IF;

END_FUNCTION_BLOCK

// ---- POUs/AutoSequence.TcPOU
FUNCTION_BLOCK AutoSequence
VAR_INPUT
END_VAR
VAR_OUTPUT
END_VAR
VAR
	
	iStep: INT;
END_VAR

// AUTO SEQUENCE
IF Memory.AutoMode THEN
CASE iStep OF
    0:  // BASIC POSITION (Home)
        // Reset all Clamps to Home Position
		Memory.RD2_OpenCmd := TRUE; Memory.RD2_CloseCmd := FALSE;
		Memory.RD1_OpenCmd := FALSE; Memory.RD1_CloseCmd := TRUE;
        Memory.CC1_Clamp_RevCmd := TRUE; Memory.CC1_Clamp_FwdCmd := FALSE;
        Memory.CC2_Clamp_RevCmd := TRUE; Memory.CC2_Clamp_FwdCmd := FALSE;
        Memory.CC3_Clamp_RevCmd := TRUE; Memory.CC3_Clamp_FwdCmd := FALSE;
        Memory.CC4_Clamp_RevCmd := TRUE; Memory.CC4_Clamp_FwdCmd := FALSE;
        Memory.CC5_Clamp_RevCmd := TRUE; Memory.CC5_Clamp_FwdCmd := FALSE;
        Memory.CC6_Clamp_RevCmd := TRUE; Memory.CC6_Clamp_FwdCmd := FALSE;
        Memory.TurnTableRevCmd:=TRUE;    Memory.TurnTableFwdCmd:=FALSE;
        // Wait for Turn Table at 0 deg (Home)
		Memory.TurnRevCmd := TRUE; Memory.TurnFwdCmd := FALSE; 
		HMI.ReadyForLoad:=TRUE;
        IF IO.TurnTableOutput.o_TurnTable_REV_SENSOR AND IO.Turn.o_Turn_REV_SENSOR AND IO.RD1.i_RD_Sensor_Close AND IO.RD2.i_RD_Sensor_Open THEN 
            iStep := 10; 
        END_IF;

    10: // LOADING PART 1 (B1-B7 & B15-B21)
        IF Memory.Stat_Parts_Lvl1_Present AND Memory.In_Operator_Outside_Cell THEN 
		
            iStep := 20;
        END_IF;

    20: // CLAMPING 1 & ROTATION (50 deg)
        IF Memory.In_PalmButton_Pushed AND  Memory.In_Operator_Outside_Cell AND IO.TurnTableOutput.o_TurnTable_REV_SENSOR AND  IO.RD1.i_RD_Sensor_Close AND IO.RD2.i_RD_Sensor_Open THEN 
            // Set Fwd, Reset Rev
            Memory.CC1_Clamp_FwdCmd := TRUE; Memory.CC1_Clamp_RevCmd := FALSE;
            Memory.CC3_Clamp_FwdCmd := TRUE; Memory.CC3_Clamp_RevCmd := FALSE;
            Memory.CC5_Clamp_FwdCmd := TRUE; Memory.CC5_Clamp_RevCmd := FALSE;
            
            // Wait for WP Feedback
            IF IO.FixtureOutput.o_CC1_CLAMPING_UNIT1_3_WP AND 
               IO.FixtureOutput.o_CC3_CLAMPING_UNIT3_3_WP AND 
               IO.FixtureOutput.o_CC5_CLAMPING_UNIT5_1_WP THEN
               
                Memory.TurnFwdCmd := TRUE; Memory.TurnRevCmd := FALSE;
                
                IF IO.Turn.o_Turn_FWD_SENSOR THEN
                    iStep := 30;
                END_IF;
            END_IF;
        END_IF;

    30: // LOADING PART 2 (B8-B14 & B22-B28)
        IF Memory.In_PalmButton_Pushed AND Memory.Stat_Parts_Lvl2_Present AND Memory.In_Operator_Outside_Cell THEN
            Memory.RD2_CloseCmd := TRUE; Memory.RD2_OpenCmd := FALSE;
            IF IO.RD2.i_RD_Sensor_Close THEN
                iStep := 40;
					HMI.ReadyForLoad:=FALSE;
            END_IF;
        END_IF;

    40: // CLAMPING 2 & WELDING CYCLE


		Memory.CC2_Clamp_FwdCmd := TRUE; Memory.CC2_Clamp_RevCmd := FALSE;
        Memory.CC4_Clamp_FwdCmd := TRUE; Memory.CC4_Clamp_RevCmd := FALSE;
        Memory.CC6_Clamp_FwdCmd := TRUE; Memory.CC6_Clamp_RevCmd := FALSE;
     
        IF IO.FixtureOutput.o_CC2_CLAMPING_UNIT2_3_WP AND
           IO.FixtureOutput.o_CC4_CLAMPING_UNIT4_3_WP AND
           IO.FixtureOutput.o_CC6_CLAMPING_UNIT6_1_WP THEN
           
            Memory.TurnTableFwdCmd := TRUE; // Start 180 deg rotation
             Memory.TurnTableRevCmd:=FALSE;
            IF WeldRobotInterface.RobotAtHome AND Memory.In_Welding_Cycle_Complete  THEN
                iStep := 50;
            END_IF;
        END_IF;

    50: // RETURN TO 0° & UNCLAMP 1
        Memory.TurnRevCmd := TRUE; Memory.TurnFwdCmd := FALSE;
        
        IF IO.Turn.o_Turn_REV_SENSOR AND  Memory.In_Welding_Cycle_Complete THEN
            // Open Part 1 Clamps
            Memory.CC1_Clamp_RevCmd := TRUE; Memory.CC1_Clamp_FwdCmd := FALSE;
            Memory.CC3_Clamp_RevCmd := TRUE; Memory.CC3_Clamp_FwdCmd := FALSE;
            Memory.CC5_Clamp_RevCmd := TRUE; Memory.CC5_Clamp_FwdCmd := FALSE;
            iStep := 60;
        END_IF;

    60: // UNLOADING PART 1
        Memory.RD1_OpenCmd := TRUE; Memory.RD1_CloseCmd := FALSE;
        
        IF IO.RD1.i_RD_Sensor_Open THEN
             Memory.Out_Robot_Start_Unload_1 := TRUE;
            IF NOT Memory.Stat_Parts_Lvl1_Present THEN
                Memory.Out_Robot_Start_Unload_1 := FALSE; // Reset Robot Request
                iStep := 70;
            END_IF;
        END_IF;

    70: // ROTATE & UNLOAD PART 2
        Memory.TurnFwdCmd := TRUE; Memory.TurnRevCmd := FALSE;
        
        IF IO.Turn.o_Turn_FWD_SENSOR THEN
            // Open Part 2 Clamps
            Memory.CC2_Clamp_RevCmd := TRUE; Memory.CC2_Clamp_FwdCmd := FALSE;
            Memory.CC4_Clamp_RevCmd := TRUE; Memory.CC4_Clamp_FwdCmd := FALSE;
            Memory.CC6_Clamp_RevCmd := TRUE; Memory.CC6_Clamp_FwdCmd := FALSE;
            
            Memory.Out_Robot_Start_Unload_2 := TRUE;
            
            IF NOT Memory.Stat_Parts_Lvl2_Present THEN
                Memory.Out_Robot_Start_Unload_2 := FALSE; // Reset Robot Request
                iStep := 0; // Cycle Finished
            END_IF;
        END_IF;

END_CASE;
ELSE
    // Manual mode logic
    Memory.CC1_Clamp_FwdCmd := HMI.CC1_Clamp_FwdCmd  ;
    Memory.CC1_Clamp_RevCmd :=HMI.CC1_Clamp_RevCmd OR HMI.Home;
	Memory.CC2_Clamp_FwdCmd := HMI.CC2_Clamp_FwdCmd;
    Memory.CC2_Clamp_RevCmd :=HMI.CC2_Clamp_RevCmd OR HMI.Home;
	Memory.CC3_Clamp_FwdCmd := HMI.CC3_Clamp_FwdCmd;
    Memory.CC3_Clamp_RevCmd :=HMI.CC3_Clamp_RevCmd OR HMI.Home;
	Memory.CC4_Clamp_FwdCmd := HMI.CC4_Clamp_FwdCmd;
    Memory.CC4_Clamp_RevCmd :=HMI.CC4_Clamp_RevCmd OR HMI.Home;
	Memory.CC5_Clamp_FwdCmd := HMI.CC5_Clamp_FwdCmd;
    Memory.CC5_Clamp_RevCmd :=HMI.CC5_Clamp_RevCmd OR HMI.Home;
	Memory.CC6_Clamp_FwdCmd := HMI.CC6_Clamp_FwdCmd;
    Memory.CC6_Clamp_RevCmd :=HMI.CC6_Clamp_RevCmd OR HMI.Home;
	Memory.RD1_OpenCmd := HMI.RD1_OpenCmd;
    Memory.RD1_CloseCmd := HMI.RD1_CloseCmd OR HMI.Home;
	
    Memory.RD2_OpenCmd := HMI.RD2_OpenCmd OR HMI.Home;
    Memory.RD2_CloseCmd := HMI.RD2_CloseCmd;
	 Memory.TurnTableFwdCmd := HMI.TurnTableFwdCmd;
    Memory.TurnTableRevCmd := HMI.TurnTableRevCmd OR HMI.Home;
	Memory.TurnTableRef:=HMI.TurnTableRef;
    Memory.TurnFwdCmd := HMI.TurnFwdCmd;
    Memory.TurnRevCmd := HMI.TurnRevCmd OR HMI.Home;
	Memory.TurnRef:=HMI.TurnRef;
    IF HMI.Home THEN
	
 iStep := 0; // reset state machine to idle
	END_IF;
END_IF;

END_FUNCTION_BLOCK

// ---- POUs/WeldRobot.TcPOU
FUNCTION_BLOCK WeldRobot
VAR_INPUT
END_VAR
VAR_OUTPUT
END_VAR
VAR
	nState: INT;
	tWeldStart: TON;
	tWeldDuration: TON;
	tReturnHome: TON;
END_VAR

IF Memory.AutoMode THEN
CASE nState OF
    0: (* WAIT FOR PART & PERMISSION *)

        IF IO.RD2.i_RD_Sensor_Close AND IO.TurnTableOutput.o_TurnTable_FWD_SENSOR AND (Memory.Stat_Parts_Lvl1_Present AND Memory.Stat_Parts_Lvl2_Present) AND Memory.AllClampWP THEN
				Memory.In_Welding_Cycle_Complete:=FALSE;
            WeldRobotInterface.WeldToCell.PickEnable := TRUE;
            WeldRobotInterface.WeldToCell.PickJobOK := FALSE;
            WeldRobotInterface.WeldToCell.InArea := TRUE;
            WeldRobotInterface.WeldToCell.PickDropProceed := TRUE;
            nState := 10;
        END_IF;

    10: (* JOB COMPLETE - PREPARE FOR WELD *)
        IF RobotInterface.RobotAtHome THEN
            WeldRobotInterface.WeldToCell.PickJobOK := TRUE;
            WeldRobotInterface.WeldToCell.DropJobOK := TRUE;
            nState := 20; // go to weld sequence
        END_IF;

    20: (* MOVE TO WELD POSITION *)
         WeldRobotInterface.RobotAtWeldPosition :=TRUE;
		 	WeldRobotInterface.RobotAtHome:=FALSE;
            tWeldStart(IN:=NOT tWeldStart.Q, PT:=T#5S); // short delay before weld
 IF    tWeldStart.Q THEN       
 nState := 30;
        END_IF;

    30: (* START WELDING *)
       
            WeldRobotInterface.TorchOn := TRUE;
            tWeldDuration(IN:=NOT tWeldDuration.Q, PT:=T#5S); // weld for 5 seconds
    IF  tWeldDuration.Q THEN     
  nState := 40;
     END_IF; 

    40: (* WELDING IN PROGRESS *)
       
            WeldRobotInterface.TorchOn := FALSE;
			
            tWeldDuration(IN:=FALSE);
          
		  nState := 50;
       

    50: (* RETURN HOME AFTER WELD *)
        tReturnHome(IN:= NOT tReturnHome.q, PT:=T#5S);
		WeldRobotInterface.RobotAtHome:=TRUE;
		WeldRobotInterface.RobotAtWeldPosition :=FALSE;
		Memory.In_Welding_Cycle_Complete:=TRUE;
        IF tReturnHome.Q AND NOT Memory.Out_Robot_Start_Unload_2 THEN
			
            nState := 0; // reset for next cycle
        END_IF;
END_CASE;
ELSE

// Manual homing logic
IF HMI.Home THEN
    WeldRobotInterface.RobotAtHome := TRUE;
		WeldRobotInterface.RobotAtWeldPosition :=FALSE;
		Memory.In_Welding_Cycle_Complete:=FALSE;
		      WeldRobotInterface.TorchOn := FALSE;
    nState := 0; // reset state machine to idle
END_IF;
END_IF;

END_FUNCTION_BLOCK

// ---- POUs/Clamping.TcPOU
FUNCTION_BLOCK Clamping
VAR_INPUT
END_VAR
VAR_OUTPUT
END_VAR
VAR
END_VAR


// cc1 clamp 1_3
IF Memory.CC1_Clamp_FwdCmd THEN
    Memory.CC1_Clamp_Rev := FALSE;
ELSIF Memory.CC1_Clamp_RevCmd THEN
    Memory.CC1_Clamp_Fwd := FALSE;
END_IF;

IF IO.FixtureOutput.o_CC1_CLAMPING_UNIT1_3_WP THEN
    Memory.CC1_Clamp_Fwd := TRUE;
END_IF;

IF IO.FixtureOutput.o_CC1_CLAMPING_UNIT1_3_HP THEN
    Memory.CC1_Clamp_Rev := TRUE;
END_IF;

// cc2 clamp 2_3
IF Memory.CC2_Clamp_FwdCmd THEN
    Memory.CC2_Clamp_Rev := FALSE;
ELSIF Memory.CC2_Clamp_RevCmd THEN
    Memory.CC2_Clamp_Fwd := FALSE;
END_IF;

IF IO.FixtureOutput.o_CC2_CLAMPING_UNIT2_3_WP THEN
    Memory.CC2_Clamp_Fwd := TRUE;
END_IF;

IF IO.FixtureOutput.o_CC2_CLAMPING_UNIT2_3_HP THEN
    Memory.CC2_Clamp_Rev := TRUE;
END_IF;

// cc3 clamp 3_3
IF Memory.CC3_Clamp_FwdCmd THEN
    Memory.CC3_Clamp_Rev := FALSE;
ELSIF Memory.CC3_Clamp_RevCmd THEN
    Memory.CC3_Clamp_Fwd := FALSE;
END_IF;

IF IO.FixtureOutput.o_CC3_CLAMPING_UNIT3_3_WP THEN
    Memory.CC3_Clamp_Fwd := TRUE;
END_IF;

IF IO.FixtureOutput.o_CC3_CLAMPING_UNIT3_3_HP THEN
    Memory.CC3_Clamp_Rev := TRUE;
END_IF;

// cc4 clamp 4_3
IF Memory.CC4_Clamp_FwdCmd THEN
    Memory.CC4_Clamp_Rev := FALSE;
ELSIF Memory.CC4_Clamp_RevCmd THEN
    Memory.CC4_Clamp_Fwd := FALSE;
END_IF;

IF IO.FixtureOutput.o_CC4_CLAMPING_UNIT4_3_WP THEN
    Memory.CC4_Clamp_Fwd := TRUE;
END_IF;

IF IO.FixtureOutput.o_CC4_CLAMPING_UNIT4_3_HP THEN
    Memory.CC4_Clamp_Rev := TRUE;
END_IF;

// CC5 clamp 5_1
IF Memory.CC5_Clamp_FwdCmd THEN
    Memory.CC5_Clamp_Rev := FALSE;
ELSIF Memory.CC5_Clamp_RevCmd THEN
    Memory.CC5_Clamp_Fwd := FALSE;
END_IF;

IF IO.FixtureOutput.o_CC5_CLAMPING_UNIT5_1_WP THEN
    Memory.CC5_Clamp_Fwd := TRUE;
END_IF;

IF IO.FixtureOutput.o_CC5_CLAMPING_UNIT5_1_HP THEN
    Memory.CC5_Clamp_Rev := TRUE;
END_IF;

// CC6 clamp 6_1
IF Memory.CC6_Clamp_FwdCmd THEN
    Memory.CC6_Clamp_Rev := FALSE;
ELSIF Memory.CC6_Clamp_RevCmd THEN
    Memory.CC6_Clamp_Fwd := FALSE;
END_IF;

IF IO.FixtureOutput.o_CC6_CLAMPING_UNIT6_1_WP THEN
    Memory.CC6_Clamp_Fwd := TRUE;
END_IF;

IF IO.FixtureOutput.o_CC6_CLAMPING_UNIT6_1_HP THEN
    Memory.CC6_Clamp_Rev := TRUE;
END_IF;

END_FUNCTION_BLOCK

// ---- POUs/vishalTest.TcPOU
FUNCTION_BLOCK vishalTest
VAR_INPUT
END_VAR
VAR_OUTPUT
END_VAR
VAR
END_VAR

END_FUNCTION_BLOCK

// ---- GlobalTextList.TcGTLO
TEXTLIST GlobalTextList
  253 = 'AirDry'
  661 = 'Auto'
  592 = 'BrushClean'
  92 = 'CC1 Clamp Fwd'
  622 = 'CC1 Clamp Fwd Work'
  495 = 'CC1 Clamp Rev Home'
  362 = 'CC2 Clamp Fwd Work'
  8 = 'CC2 Clamp Rev Home'
  326 = 'CC3 Clamp Fwd Work'
  960 = 'CC3 Clamp Rev Home'
  425 = 'CC4 Clamp Fwd Work'
  39 = 'CC4 Clamp Rev Home'
  420 = 'CC5 Clamp Fwd Work'
  194 = 'CC5 Clamp Rev Home'
  327 = 'CC6 Clamp Fwd Work'
  248 = 'CC6 Clamp Rev Home'
  497 = 'Drop Comp'
  774 = 'Gripper Close'
  168 = 'Gripper Open'
  467 = 'Home'
  950 = 'OP Load'
  321 = 'Palm Button'
  648 = 'Part Present 1'
  395 = 'Part Present 2'
  60 = 'RD1 Close'
  135 = 'RD1 Fwd Open'
  347 = 'RD1 Open'
  466 = 'RD2 Close'
  546 = 'RD2 Open'
  715 = 'READY FOR LOAD'
  165 = 'RinseSpray'
  367 = 'Robot At weld'
  734 = 'Robot Pick'
  454 = 'RobotAtHome'
  127 = 'SoapSpray'
  652 = 'TT Fwd 180 Work'
  191 = 'TT Fwd Work'
  849 = 'TT Reference'
  781 = 'TT Rev 0 Home'
  468 = 'TT Rev Home'
  563 = 'Turn 0deg Home'
  647 = 'Turn 50deg Work'
  794 = 'Turn 70deg Work'
  596 = 'Turn Fwd Work'
  9 = 'Turn Reference'
  884 = 'Turn Rev Home'
  928 = 'WaterSpray'
  871 = 'Weld Comp'
  159 = 'Weld Comp['
  755 = 'Weld On'
  122 = 'WeldComp'
END_TEXTLIST

// ---- VISUs/Clamp.TcVIS
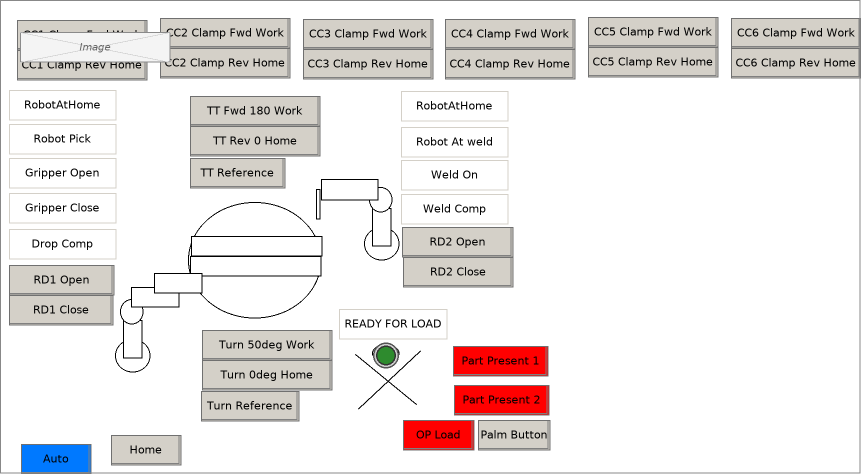
VISUALIZATION Clamp  // 861x474
    Button (17,20 130x30), "CC1 Clamp Fwd Work", colour toggle: IO.FixtureOutput.o_CC1_CLAMPING_UNIT1_3_WP
        tap HMI.CC1_Clamp_FwdCmd
    Button (17,50 130x30), "CC1 Clamp Rev Home", colour toggle: IO.FixtureOutput.o_CC1_CLAMPING_UNIT1_3_HP
        tap HMI.CC1_Clamp_RevCmd
    Button (160,18 130x30), "CC2 Clamp Fwd Work", colour toggle: IO.FixtureOutput.o_CC2_CLAMPING_UNIT2_3_WP
        tap HMI.CC2_Clamp_FwdCmd
    Button (160,48 130x30), "CC2 Clamp Rev Home", colour toggle: IO.FixtureOutput.o_CC2_CLAMPING_UNIT2_3_HP
        tap HMI.CC2_Clamp_RevCmd
    Button (303,19 130x30), "CC3 Clamp Fwd Work", colour toggle: IO.FixtureOutput.o_CC3_CLAMPING_UNIT3_3_WP
        tap HMI.CC3_Clamp_FwdCmd
    Button (303,49 130x30), "CC3 Clamp Rev Home", colour toggle: IO.FixtureOutput.o_CC3_CLAMPING_UNIT3_3_HP
        tap HMI.CC3_Clamp_RevCmd
    Button (445,19 130x30), "CC4 Clamp Fwd Work", colour toggle: IO.FixtureOutput.o_CC4_CLAMPING_UNIT4_3_WP
        tap HMI.CC4_Clamp_FwdCmd
    Button (445,49 130x30), "CC4 Clamp Rev Home", colour toggle: IO.FixtureOutput.o_CC4_CLAMPING_UNIT4_3_HP
        tap HMI.CC4_Clamp_RevCmd
    Button (588,17 130x30), "CC5 Clamp Fwd Work", colour toggle: IO.FixtureOutput.o_CC5_CLAMPING_UNIT5_1_WP
        tap HMI.CC5_Clamp_FwdCmd
    Button (588,47 130x30), "CC5 Clamp Rev Home", colour toggle: IO.FixtureOutput.o_CC5_CLAMPING_UNIT5_1_HP
        tap HMI.CC5_Clamp_RevCmd
    Button (731,18 130x30), "CC6 Clamp Fwd Work", colour toggle: IO.FixtureOutput.o_CC6_CLAMPING_UNIT6_1_WP
        tap HMI.CC6_Clamp_FwdCmd
    Button (731,48 130x30), "CC6 Clamp Rev Home", colour toggle: IO.FixtureOutput.o_CC6_CLAMPING_UNIT6_1_HP
        tap HMI.CC6_Clamp_RevCmd
    Button (9,265 105x30), "RD1 Open", colour toggle: IO.RD1.i_RD_Sensor_Open
        tap HMI.RD1_OpenCmd
    Button (9,295 104x30), "RD1 Close", colour toggle: IO.RD1.i_RD_Sensor_Close
        tap HMI.RD1_CloseCmd
    Button (402,227 111x30), "RD2 Open", colour toggle: IO.RD2.i_RD_Sensor_Open
        tap HMI.RD2_OpenCmd
    Button (403,257 110x30), "RD2 Close", colour toggle: IO.RD2.i_RD_Sensor_Close
        tap HMI.RD2_CloseCmd
    Button (190,96 130x30), "TT Fwd 180 Work", colour toggle: IO.TurnTableOutput.o_TurnTable_FWD_SENSOR
        tap HMI.TurnTableFwdCmd
    Button (190,126 130x30), "TT Rev 0 Home", colour toggle: IO.TurnTableOutput.o_TurnTable_REV_SENSOR
        tap HMI.TurnTableRevCmd
    Button (190,158 95x30), "TT Reference", colour toggle: IO.TurnTableOutput.o_TurnTable_REF_SENSOR
        tap HMI.TurnTableRef
    Ellipse (188,202 133x116)
    Button (202,330 130x30), "Turn 50deg Work", colour toggle: IO.Turn.o_Turn_FWD_SENSOR
        tap HMI.TurnFwdCmd
    Button (202,360 130x30), "Turn 0deg Home", colour toggle: IO.Turn.o_Turn_REV_SENSOR
        tap HMI.TurnRevCmd
    Button (201,391 98x30), "Turn Reference", colour toggle: IO.Turn.o_Turn_REF_SENSOR
        tap HMI.TurnRef
    Rectangle (190,256 131x20), colour toggle: Memory.Stat_Parts_Lvl2_Present
    Ellipse (372,344 27x18)
    Line (355,354) (416,404)
    Line (420,351) (358,409)
    Image (20,32 150x30)
    Button (403,420 71x30), "OP Load", colour toggle: Memory.In_Operator_Outside_Cell
        toggle Memory.In_Operator_Outside_Cell
    Button (453,346 95x30), "Part Present 1", colour toggle: Memory.Stat_Parts_Lvl1_Present
        toggle Memory.Stat_Parts_Lvl1_Present
    Button (454,385 95x30), "Part Present 2", colour toggle: Memory.Stat_Parts_Lvl2_Present
        toggle Memory.Stat_Parts_Lvl2_Present
    Button (478,420 72x30), "Palm Button", colour toggle: Memory.In_PalmButton_Pushed
        tap Memory.In_PalmButton_Pushed
    Button (21,444 70x30), "Auto", colour toggle: Memory.AutoMode
        toggle Memory.AutoMode
    Button (111,435 70x30), "Home", colour toggle: HMI.Home
        tap HMI.Home
    Ellipse (115,339 35x33)
    Rectangle (123,320 19x38)
    Ellipse (120,299 23x25)
    Rectangle (131,287 48x20), angle 331
    Rectangle (154,273 48x20), angle 236, colour toggle: RobotInterface.HDL_HandlingToCell.Gripper1ClosedAck
    Ellipse (364,227 35x33)
    Rectangle (372,208 19x38)
    Ellipse (369,187 23x25)
    Rectangle (321,179 57x21), angle 13
    Rectangle (316,189 4x30), angle 17, colour toggle: WeldRobotInterface.TorchOn
    Lamp1 (371,338 30x35), variable: HMI.ReadyForLoad, style: Lamp-Lamp1-Green
    Textfield (339,309 108x30), "READY FOR LOAD"
    Textfield (9,90 107x30), "RobotAtHome", text variable: RobotInterface.RobotAtHome, colour toggle: RobotInterface.RobotAtHome
    Textfield (9,124 107x30), "Robot Pick", text variable: RobotInterface.HDL_HandlingToCell.PickJobProceed, colour toggle: RobotInterface.HDL_HandlingToCell.PickJobProceed
    Textfield (9,158 107x30), "Gripper Open", text variable: RobotInterface.HDL_HandlingToCell.Gripper1OpenedAck, colour toggle: RobotInterface.HDL_HandlingToCell.Gripper1OpenedAck
    Textfield (9,193 107x30), "Gripper Close", text variable: RobotInterface.HDL_HandlingToCell.Gripper1ClosedAck, colour toggle: RobotInterface.HDL_HandlingToCell.Gripper1ClosedAck
    Textfield (9,229 107x30), "Drop Comp", text variable: RobotInterface.HDL_HandlingToCell.DropJobProceed, colour toggle: RobotInterface.HDL_HandlingToCell.PickJobOK
    Textfield (401,91 107x30), "RobotAtHome", text variable: WeldRobotInterface.RobotAtHome, colour toggle: WeldRobotInterface.RobotAtHome
    Textfield (401,160 107x30), "Weld On", text variable: WeldRobotInterface.TorchOn, colour toggle: WeldRobotInterface.TorchOn
    Textfield (401,127 107x30), "Robot At weld", text variable: WeldRobotInterface.RobotAtWeldPosition, colour toggle: WeldRobotInterface.RobotAtWeldPosition
    Textfield (401,194 107x30), "Weld Comp", text variable: Memory.In_Welding_Cycle_Complete, colour toggle: Memory.In_Welding_Cycle_Complete
    Rectangle (191,236 131x20), colour toggle: Memory.Stat_Parts_Lvl1_Present
END_VISUALIZATION
